PROGRAM MAIN
VAR
		bStartStop	:BOOL;
		nCounter	:DINT;
END_VAR

IF bStartStop THEN
	nCounter	:= nCounter + 1;
END_IF

END_PROGRAM

(* stored: Version 1.1.0.1, ProductVersion 3.1.4024.2
   POU MAIN: Id {6321da77-73e8-4248-948c-17bbd0ea002d}, SpecialFunc None *)
